TYPE RunningStates :
(	
	Start,
	Preparation,
	WarmUp,
	Running,
	EndRun
	) := Start;
END_TYPE

(* stored: Version 1.1.0.1, ProductVersion 3.1.4024.15
   DUT RunningStates: Id {ca075d44-347a-4c24-a521-7a9b74f5dba5} *)
